// TIA Portal V17 export
// export: Created 2022-02-03T14:45:16.1562038Z, ExportSetting WithDefaults, DisplayName Totally Integrated Automation Portal, DisplayVersion V17, DisplayName TIA Portal Openness, DisplayVersion V17, DisplayName TIA Portal Version Control Interface, DisplayVersion V17, DisplayName SINAMICS Startdrive Advanced, DisplayVersion V17, DisplayName SINAMICS Startdrive G130, G150, S120, S150, SINAMICS MV, S210, DisplayVersion V17, DisplayName SINAMICS Startdrive G110M, G120, G120C, G120D, G120P, G115D, DisplayVersion V17, DisplayName STEP 7 Professional, DisplayVersion V17, DisplayName STEP 7 Safety, DisplayVersion V17, DisplayName WinCC Advanced, DisplayVersion V17
DATA_BLOCK "interfaceTP"   // DB3
VERSION : 0.1
// stored: Access Published, AutoNumber true, DBAccessibleFromOPCUA true
   VAR
      operationMode : Bool;
      operationMan : Bool;
      operationAuto : Bool;
      sequencerMode : Bool;
      jogRight : Bool;
      jogLeft : Bool;
      conveyorFault : Bool;
      acknowledgeFault : Bool;
      storeNo : UInt;
      currentStoreFull : Bool;
      initCurrentStore : Bool;
      initAllStores : Bool;
      IODeviceError : Bool;
      IODeviceNo : Int;
      IODeviceSlotNo : Int;
      messageBits : Word;
      weightAt : "TypeWeights";
      statistics { S7_SetPoint := 'True'} : "typeStatistics";
   END_VAR
   VAR RETAIN
      storeStatistics { S7_SetPoint := 'True'} : "typeStoreStatistics";
   END_VAR
   VAR
      deviceFail { S7_SetPoint := 'True'} : LDT;
      deviceReturn : LDT;
      failDuration : LTime;
   END_VAR
BEGIN
END_DATA_BLOCK
